// TIA Portal V19 export
DATA_BLOCK "AI SCALING DB"   // DB5
{ S7_Optimized_Access := 'FALSE' }
   VAR
      MIN : Struct
         "LEVEL TRANSMITTER-101 ANALOG" : Real := 0.0;
         "LEVEL TRANSMITTER-102 ANALOG" : Real := 0.0;
         "DIFFRENTIAL PRESSURE TRANSMITTER-101 ANALOG" : Real := 0.0;
         "CONDUCTIVITY INDICATOR CUM TRANSMITTER-101" : Real := 0.0;
         "DIFFRENTIAL PRESSURE TRANSMITTER-201" : Real := 0.0;
         "FLOW INDICATIOR TOTALISER-201" : Real := 0.0;
         "LEVEL TRANSMITTER-201" : Real := 0.0;
         "LEVEL TRANSMITTER-801" : Real := 0.0;
         "RESISTIVITY CUM TRANSMITTER 601" { S7_SetPoint := 'True'} : Real := 0.0;
         "PRESSURE TRANSMITTER 601" { S7_SetPoint := 'True'} : Real := 0.0;
         "FLOW INDICATIOR TOTALISER 601" { S7_SetPoint := 'True'} : Real := 0.0;
         "PH INDICATOR CUM TRANSMITTER 601" { S7_SetPoint := 'True'} : Real := 0.0;
         "UV-601_SENSOR" { S7_SetPoint := 'True'} : Real := 0.0;
         "SPARE(30)" { S7_SetPoint := 'True'} : Real := 0.0;
         "SPARE(31)" { S7_SetPoint := 'True'} : Real := 0.0;
         "SPARE(32)" { S7_SetPoint := 'True'} : Real := 0.0;
      END_STRUCT;
      MAX : Struct
         "LEVEL TRANSMITTER-101 ANALOG" { S7_SetPoint := 'True'} : Real := 100.0;
         "LEVEL TRANSMITTER-102 ANALOG" { S7_SetPoint := 'True'} : Real := 100.0;
         "DIFFRENTIAL PRESSURE TRANSMITTER-101 ANALOG" { S7_SetPoint := 'True'} : Real := 2.0;
         "CONDUCTIVITY INDICATOR CUM TRANSMITTER-101" { S7_SetPoint := 'True'} : Real := 1999.0;
         "DIFFRENTIAL PRESSURE TRANSMITTER-201" { S7_SetPoint := 'True'} : Real := 2.0;
         "FLOW INDICATIOR TOTALISER-201" { S7_SetPoint := 'True'} : Real := 20.0;
         "LEVEL TRANSMITTER-201" { S7_SetPoint := 'True'} : Real := 100.0;
         "LEVEL TRANSMITTER-801" { S7_SetPoint := 'True'} : Real := 100.0;
         "RESISTIVITY CUM TRANSMITTER 601" { S7_SetPoint := 'True'} : Real := 100.0;
         "PRESSURE TRANSMITTER 601" { S7_SetPoint := 'True'} : Real := 10.0;
         "FLOW INDICATIOR TOTALISER 601" { S7_SetPoint := 'True'} : Real := 56.0;
         "PH INDICATOR CUM TRANSMITTER 601" { S7_SetPoint := 'True'} : Real := 14.0;
         "UV-601_SENSOR" { S7_SetPoint := 'True'} : Real := 120.0;
         "SPARE(30)" { S7_SetPoint := 'True'} : Real;
         "SPARE(31)" { S7_SetPoint := 'True'} : Real;
         "SPARE(32)" { S7_SetPoint := 'True'} : Real;
      END_STRUCT;
      PV : Struct
         "LEVEL TRANSMITTER-101 ANALOG" : Real;
         "LEVEL TRANSMITTER-102 ANALOG" : Real;
         "DIFFRENTIAL PRESSURE TRANSMITTER-101 ANALOG" : Real;
         "CONDUCTIVITY INDICATOR CUM TRANSMITTER-101" : Real;
         "DIFFRENTIAL PRESSURE TRANSMITTER-201" : Real;
         "FLOW INDICATIOR TOTALISER-201" : Real;
         "LEVEL TRANSMITTER-201" : Real;
         "LEVEL TRANSMITTER-801" : Real;
         "RESISTIVITY CUM TRANSMITTER 601" : Real;
         "PRESSURE TRANSMITTER 601" : Real;
         "FLOW INDICATIOR TOTALISER 601" : Real;
         "PH INDICATOR CUM TRANSMITTER 601" : Real;
         "UV-601_SENSOR" : Real;
         "SPARE(30)" : Real;
         "SPARE(31)" : Real;
         "SPARE(32)" : Real;
      END_STRUCT;
      SPARE : Bool;
      "LT-101" : Struct
         LOW_BUFF : Int;
         HIGH_BUFF : Int;
      END_STRUCT;
      "LT-102" : Struct
         LOW_BUFF : Int;
         HIGH_BUFF : Int;
      END_STRUCT;
      "LT-201" : Struct
         LOW_BUFF : Int;
         HIGH_BUFF : Int;
      END_STRUCT;
      "LT-801" : Struct
         LOW_BUFF : Int;
         HIGH_BUFF : Int;
      END_STRUCT;
      "LT-101 SET VALVE" : Struct
         LL : Real;
         L : Real;
         H : Real;
         HH : Real;
      END_STRUCT;
      "LT-102 SET VALVE" : Struct
         LL : Real;
         L : Real;
         H : Real;
         HH : Real;
      END_STRUCT;
      "LT-201 SET VALVE" : Struct
         LL : Real;
         L : Real;
         H : Real;
         HH : Real;
      END_STRUCT;
      "LT-801 SET VALVE" : Struct
         LL : Real;
         L : Real;
         H : Real;
         HH : Real;
      END_STRUCT;
   END_VAR
BEGIN
END_DATA_BLOCK
